    rq_activate_all_grippers(False)
    # end: URCap Program Node
    $ 4 "MoveJ"
    $ 5 "Waypoint_2" "breakAfter"
    movej(get_inverse_kin(Waypoint_2_p, qnear=Waypoint_2_q), a=1.3962634015954636, v=1.0471975511965976)
    $ 6 "Wait sensor=LO"
    while (get_standard_digital_in(0) == True):
      sync()
    end
    $ 7 "Pallet_1"
    def Pallet_1_trans(pose):
    return p[pose[0], pose[1], pose[2], 0, 0, 0]
  end
  def Pallet_1_rot(pose):
  return p[0, 0, 0, pose[3], pose[4], pose[5]]
  end
  def Pallet_1_compute_pallet_waypoint(T_base_feature_taught, T_feature_referencePoint_taught, T_referencePoint_approach_taught, T_base_feature, T_base_referencePoint):
  local trans_referencePoint_approach_in_feature_taught = pose_sub(Pallet_1_trans(pose_trans(T_feature_referencePoint_taught, T_referencePoint_approach_taught)), Pallet_1_trans(T_feature_referencePoint_taught))
  local rot_referencePoint_approach_in_feature_taught = pose_trans(Pallet_1_rot(T_feature_referencePoint_taught), pose_trans(Pallet_1_rot(T_referencePoint_approach_taught), pose_inv(Pallet_1_rot(T_feature_referencePoint_taught))))
  T_feature_referencePoint = pose_trans(pose_inv(T_base_feature), T_base_referencePoint)
  rot_referencePoint_approach = pose_trans(pose_inv(Pallet_1_rot(T_feature_referencePoint)), pose_trans(rot_referencePoint_approach_in_feature_taught, Pallet_1_rot(T_feature_referencePoint)))
  T_feature_approach = pose_trans(trans_referencePoint_approach_in_feature_taught, pose_trans(T_feature_referencePoint, rot_referencePoint_approach))
  T_base_approach = pose_trans(T_base_feature, T_feature_approach)
  return T_base_approach
  end
  Pallet_1_tct = 1
  if (Pallet_1_cnt_1 > 1 or Pallet_1_cnt_1 < 1):
    Pallet_1_cnt_1 = 1
  end
  $ 8 "Patterns" "noBreak"
  $ 9 "Irreg_Pattern_1" "noBreak"
  $ 11 "Layers" "noBreak"
  if (Pallet_1_cnt_1 < 2):
    Pallet_1_lno = 1
    Pallet_1_lct = Pallet_1_cnt_1
    global Item_1=pose_trans(p[0.0,0.0,0.0,0.0,0.0,0.0], pose_trans(p[-.000000000000, -.000000000000, -.000000000000, .000000000000, .000000000000, .000000000000], p[-.338171139538, -.420737183303, .092764235338, .009876315371, -3.096236515232, .249936558774]))
    if ((Pallet_1_lct - 1) == 0):
      referencePoint = Item_1
      Waypoint_6_q = [0.5956683158844361, -0.6755548280618635, 0.603014294320757, -1.6180516682204722, -1.4727962652724997, -0.9768632094038221]
    end
    direction = p[0,0,1,0,0,0]
    referencePoint = pose_add (referencePoint,p[0.0*direction[0],0.0*direction[1],0.0*direction[2],0,0,0])
  end
  Waypoint_6_p = Pallet_1_compute_pallet_waypoint(p[0.0,0.0,0.0,0.0,0.0,0.0], pose_trans(pose_inv(p[0.0,0.0,0.0,0.0,0.0,0.0]), p[-0.35656855679907695,-0.4237765193480358,0.0916497228884191,0.14229659831444877,-3.021243201222635,0.176167743332585]), p[-0.050081541706238464,-0.002934815571442262,-0.05522053959512324,0.06280827340026365,0.001341962689266323,0.110632066395465], p[0.0,0.0,0.0,0.0,0.0,0.0], referencePoint)
  Waypoint_6_p = pose_trans(p[-0.35656855679907695,-0.4237765193480358,0.0916497228884191,0.14229659831444882,-3.021243201222637,0.17616774333258506], pose_trans(pose_inv(referencePoint), Waypoint_6_p))
  Waypoint_7_p = Pallet_1_compute_pallet_waypoint(p[0.0,0.0,0.0,0.0,0.0,0.0], pose_trans(pose_inv(p[0.0,0.0,0.0,0.0,0.0,0.0]), p[-0.35656855679907695,-0.4237765193480358,0.0916497228884191,0.14229659831444877,-3.021243201222635,0.176167743332585]), p[-0.0972432192339368,0.006486004980699234,-0.006903856687141913,-0.09058990540327166,-0.07880304154291709,0.12847659139677955], p[0.0,0.0,0.0,0.0,0.0,0.0], referencePoint)
  Waypoint_7_p = pose_trans(p[-0.35656855679907695,-0.4237765193480358,0.0916497228884191,0.14229659831444882,-3.021243201222637,0.17616774333258506], pose_trans(pose_inv(referencePoint), Waypoint_7_p))
  Waypoint_6_p = Pallet_1_compute_pallet_waypoint(p[0.0,0.0,0.0,0.0,0.0,0.0], pose_trans(pose_inv(p[0.0,0.0,0.0,0.0,0.0,0.0]), p[-0.35656855679907695,-0.4237765193480358,0.0916497228884191,0.14229659831444877,-3.021243201222635,0.176167743332585]), p[-0.050081541706238464,-0.002934815571442262,-0.05522053959512324,0.06280827340026365,0.001341962689266323,0.110632066395465], p[0.0,0.0,0.0,0.0,0.0,0.0], referencePoint)
  Waypoint_6_p = pose_trans(p[-0.35656855679907695,-0.4237765193480358,0.0916497228884191,0.14229659831444882,-3.021243201222637,0.17616774333258506], pose_trans(pose_inv(referencePoint), Waypoint_6_p))
  $ 12 "At Each Item" "noBreak"
  $ 13 "Generated Movements" "noBreak"
  $ 14 "MoveJ" "noBreak"
  $ 15 "Waypoint_6" "noBreak"
  movej(get_inverse_kin(pose_trans(referencePoint, pose_trans(p[-.400294158776, .393560298227, .001491262390, -.142296598314, 3.021243201223, -.176167743333], Waypoint_6_p)), qnear=Waypoint_6_q), a=1.3962634015954636, v=1.0471975511965976)
  $ 16 "MoveL" "noBreak"
  $ 17 "Waypoint_7" "noBreak"
  movel(pose_trans(referencePoint, pose_trans(p[-.400294158776, .393560298227, .001491262390, -.142296598314, 3.021243201223, -.176167743333], Waypoint_7_p)), a=1.2, v=0.25)
  $ 18 "Set Payload: Payload" "noBreak"
  set_target_payload(0.450000, [0.000000, 0.000000, 0.000000], [0.000407, 0.000407, 0.000407, 0.000000, 0.000000, 0.000000])
  $ 19 "Tool action" "noBreak"
  # begin: URCap Program Node
  #   Source: Robotiq_Grippers, 2.4.0.45103, Robotiq Inc.
  #   Type: Gripper
  $ 20 "Gripper Close (3)" "noBreak"
  if not(gripper_connected[2]):
    popup("Gripper 3 must be connected to run this program.", "No connection", False, True, True)
  end
  if not(rq_is_gripper_activated("3")):
    popup("Gripper 3 is not activated. Go to Installation tab > Gripper to activate it and run the program again.", "Not activated", False, True, True)
  end
  rq_set_pos_spd_for(255, 255, 13, "3")
  rq_wait_pos_spe_for_request(255, 255, 13, "3")
  rq_go_to("3")
  rq_wait("3")
  # end: URCap Program Node
  $ 21 "MoveL" "noBreak"
  $ 22 "Waypoint_6" "noBreak"
  movel(pose_trans(referencePoint, pose_trans(p[-.400294158776, .393560298227, .001491262390, -.142296598314, 3.021243201223, -.176167743333], Waypoint_6_p)), a=1.2, v=0.25)
  Pallet_1_sep = False
  if (Pallet_1_cnt_1 >= 1):
    Pallet_1_cnt_1 = 1
  else:
    Pallet_1_cnt_1 = Pallet_1_cnt_1 + 1
  end
  $ 23 "Pallet_2"
  def Pallet_2_trans(pose):
  return p[pose[0], pose[1], pose[2], 0, 0, 0]
  end
  def Pallet_2_rot(pose):
  return p[0, 0, 0, pose[3], pose[4], pose[5]]
  end
  def Pallet_2_compute_pallet_waypoint(T_base_feature_taught, T_feature_referencePoint_taught, T_referencePoint_approach_taught, T_base_feature, T_base_referencePoint):
  local trans_referencePoint_approach_in_feature_taught = pose_sub(Pallet_2_trans(pose_trans(T_feature_referencePoint_taught, T_referencePoint_approach_taught)), Pallet_2_trans(T_feature_referencePoint_taught))
  local rot_referencePoint_approach_in_feature_taught = pose_trans(Pallet_2_rot(T_feature_referencePoint_taught), pose_trans(Pallet_2_rot(T_referencePoint_approach_taught), pose_inv(Pallet_2_rot(T_feature_referencePoint_taught))))
  T_feature_referencePoint = pose_trans(pose_inv(T_base_feature), T_base_referencePoint)
  rot_referencePoint_approach = pose_trans(pose_inv(Pallet_2_rot(T_feature_referencePoint)), pose_trans(rot_referencePoint_approach_in_feature_taught, Pallet_2_rot(T_feature_referencePoint)))
  T_feature_approach = pose_trans(trans_referencePoint_approach_in_feature_taught, pose_trans(T_feature_referencePoint, rot_referencePoint_approach))
  T_base_approach = pose_trans(T_base_feature, T_feature_approach)
  return T_base_approach
  end
  Pallet_2_tct = 1
  if (Pallet_2_cnt_1 > 1 or Pallet_2_cnt_1 < 1):
    Pallet_2_cnt_1 = 1
  end
  $ 24 "Patterns" "noBreak"
  $ 25 "Irreg_Pattern_2" "noBreak"
  $ 27 "Layers" "noBreak"
  if (Pallet_2_cnt_1 < 2):
    Pallet_2_lno = 1
    Pallet_2_lct = Pallet_2_cnt_1
    global Item_2=pose_trans(p[0.0,0.0,0.0,0.0,0.0,0.0], pose_trans(p[-.000000000000, -.000000000000, -.000000000000, .000000000000, .000000000000, .000000000000], p[-.463665534965, -.106220808801, .035787281560, 2.122926777319, 2.233821671100, -.100576269136]))
    if ((Pallet_2_lct - 1) == 0):
      referencePoin_1 = Item_2
      Waypoint_5_q = [-0.10132915178099822, -0.8465228837704926, 1.1239708105507988, -1.842076917673376, -1.4983623663589887, -0.15588361421827113]
    end
    direction = p[0,0,1,0,0,0]
    referencePoin_1 = pose_add (referencePoin_1,p[0.0*direction[0],0.0*direction[1],0.0*direction[2],0,0,0])
  end
  Waypoint_5_p = Pallet_2_compute_pallet_waypoint(p[0.0,0.0,0.0,0.0,0.0,0.0], pose_trans(pose_inv(p[0.0,0.0,0.0,0.0,0.0,0.0]), p[-0.4636655349654482,-0.10622080880105224,0.035787281559670425,2.1229267773186806,2.233821671099525,-0.10057626913611485]), p[0.0025464538946822213,0.007379050264824327,-0.053400380694234195,-0.03847629676856576,-0.00190489899378521,-0.0019139929032188495], p[0.0,0.0,0.0,0.0,0.0,0.0], referencePoin_1)
  Waypoint_5_p = pose_trans(p[-0.4636655349654482,-0.10622080880105224,0.035787281559670425,2.122926777318679,2.233821671099524,-0.10057626913611215], pose_trans(pose_inv(referencePoin_1), Waypoint_5_p))
  ToolActionPoi_1_p = Pallet_2_compute_pallet_waypoint(p[0.0,0.0,0.0,0.0,0.0,0.0], pose_trans(pose_inv(p[0.0,0.0,0.0,0.0,0.0,0.0]), p[-0.4636655349654482,-0.10622080880105224,0.035787281559670425,2.1229267773186806,2.233821671099525,-0.10057626913611485]), p[0.0,5.551115123125783E-17,2.7755575615628914E-17,-2.567396382296971E-12,1.8025025916301725E-12,-1.5242017175308427E-12], p[0.0,0.0,0.0,0.0,0.0,0.0], referencePoin_1)
  ToolActionPoi_1_p = pose_trans(p[-0.4636655349654482,-0.10622080880105224,0.035787281559670425,2.122926777318679,2.233821671099524,-0.10057626913611215], pose_trans(pose_inv(referencePoin_1), ToolActionPoi_1_p))
  Waypoint_5_p = Pallet_2_compute_pallet_waypoint(p[0.0,0.0,0.0,0.0,0.0,0.0], pose_trans(pose_inv(p[0.0,0.0,0.0,0.0,0.0,0.0]), p[-0.4636655349654482,-0.10622080880105224,0.035787281559670425,2.1229267773186806,2.233821671099525,-0.10057626913611485]), p[0.0025464538946822213,0.007379050264824327,-0.053400380694234195,-0.03847629676856576,-0.00190489899378521,-0.0019139929032188495], p[0.0,0.0,0.0,0.0,0.0,0.0], referencePoin_1)
  Waypoint_5_p = pose_trans(p[-0.4636655349654482,-0.10622080880105224,0.035787281559670425,2.122926777318679,2.233821671099524,-0.10057626913611215], pose_trans(pose_inv(referencePoin_1), Waypoint_5_p))
  $ 28 "At Each Item" "noBreak"
  $ 29 "Generated Movements" "noBreak"
  $ 30 "MoveJ" "noBreak"
  $ 31 "Waypoint_5" "noBreak"
  movej(get_inverse_kin(pose_trans(referencePoin_1, pose_trans(p[.085151670364, .468686561658, .025128032432, -2.122926777319, -2.233821671100, .100576269136], Waypoint_5_p)), qnear=Waypoint_5_q), a=1.3962634015954636, v=1.0471975511965976)
  $ 32 "MoveL" "noBreak"
  $ 33 "ToolActionPoi_1" "noBreak"
  movel(pose_trans(referencePoin_1, pose_trans(p[.085151670364, .468686561658, .025128032432, -2.122926777319, -2.233821671100, .100576269136], ToolActionPoi_1_p)), a=1.2, v=0.25)
  $ 34 "Tool action" "noBreak"
  # begin: URCap Program Node
  #   Source: Robotiq_Grippers, 2.4.0.45103, Robotiq Inc.
  #   Type: Gripper
  $ 35 "Gripper Open (3)" "noBreak"
  if not(gripper_connected[2]):
    popup("Gripper 3 must be connected to run this program.", "No connection", False, True, True)
  end
  if not(rq_is_gripper_activated("3")):
    popup("Gripper 3 is not activated. Go to Installation tab > Gripper to activate it and run the program again.", "Not activated", False, True, True)
  end
  rq_set_pos_spd_for(0, 255, 255, "3")
  rq_wait_pos_spe_for_request(0, 255, 255, "3")
  rq_go_to("3")
  rq_wait("3")
  # end: URCap Program Node
  $ 36 "MoveL" "noBreak"
  $ 37 "Waypoint_5" "noBreak"
  movel(pose_trans(referencePoin_1, pose_trans(p[.085151670364, .468686561658, .025128032432, -2.122926777319, -2.233821671100, .100576269136], Waypoint_5_p)), a=1.2, v=0.25)
  Pallet_2_sep = False
  if (Pallet_2_cnt_1 >= 1):
    Pallet_2_cnt_1 = 1
  else:
    Pallet_2_cnt_1 = Pallet_2_cnt_1 + 1
  end
  $ 38 "MoveL"
  $ 39 "Waypoint_1" "breakAfter"
  movel(Waypoint_1_p, a=1.2, v=0.25)
  $ 40 "Wait: 3.0"
  sleep(3.0)
  $ 41 "Pallet_3"
  def Pallet_3_trans(pose):
  return p[pose[0], pose[1], pose[2], 0, 0, 0]
  end
  def Pallet_3_rot(pose):
  return p[0, 0, 0, pose[3], pose[4], pose[5]]
  end
  def Pallet_3_compute_pallet_waypoint(T_base_feature_taught, T_feature_referencePoint_taught, T_referencePoint_approach_taught, T_base_feature, T_base_referencePoint):
  local trans_referencePoint_approach_in_feature_taught = pose_sub(Pallet_3_trans(pose_trans(T_feature_referencePoint_taught, T_referencePoint_approach_taught)), Pallet_3_trans(T_feature_referencePoint_taught))
  local rot_referencePoint_approach_in_feature_taught = pose_trans(Pallet_3_rot(T_feature_referencePoint_taught), pose_trans(Pallet_3_rot(T_referencePoint_approach_taught), pose_inv(Pallet_3_rot(T_feature_referencePoint_taught))))
  T_feature_referencePoint = pose_trans(pose_inv(T_base_feature), T_base_referencePoint)
  rot_referencePoint_approach = pose_trans(pose_inv(Pallet_3_rot(T_feature_referencePoint)), pose_trans(rot_referencePoint_approach_in_feature_taught, Pallet_3_rot(T_feature_referencePoint)))
  T_feature_approach = pose_trans(trans_referencePoint_approach_in_feature_taught, pose_trans(T_feature_referencePoint, rot_referencePoint_approach))
  T_base_approach = pose_trans(T_base_feature, T_feature_approach)
  return T_base_approach
  end
  Pallet_2_tct_1 = 1
  if (Pallet_2_cnt_2 > 1 or Pallet_2_cnt_2 < 1):
    Pallet_2_cnt_2 = 1
  end
  $ 42 "Patterns" "noBreak"
  $ 43 "Irreg_Pattern_3" "noBreak"
  $ 45 "Layers" "noBreak"
  if (Pallet_2_cnt_2 < 2):
    Pallet_2_lno_1 = 1
    Pallet_2_lct_1 = Pallet_2_cnt_2
    global Item_3=pose_trans(p[0.0,0.0,0.0,0.0,0.0,0.0], pose_trans(p[-.000000000000, -.000000000000, -.000000000000, .000000000000, .000000000000, .000000000000], p[-.463665534965, -.106220808801, .035787281560, 2.122926777319, 2.233821671100, -.100576269136]))
    if ((Pallet_2_lct_1 - 1) == 0):
      referencePoin_2 = Item_3
      Waypoint_5_q = [-0.10132915178099822, -0.8465228837704926, 1.1239708105507988, -1.842076917673376, -1.4983623663589887, -0.15588361421827113]
    end
    direction = p[0,0,1,0,0,0]
    referencePoin_2 = pose_add (referencePoin_2,p[0.0*direction[0],0.0*direction[1],0.0*direction[2],0,0,0])
  end
  Waypoint_5_p = Pallet_3_compute_pallet_waypoint(p[0.0,0.0,0.0,0.0,0.0,0.0], pose_trans(pose_inv(p[0.0,0.0,0.0,0.0,0.0,0.0]), p[-0.4636655349654482,-0.10622080880105224,0.035787281559670425,2.1229267773186806,2.233821671099525,-0.10057626913611485]), p[0.0025464538946822213,0.007379050264824327,-0.053400380694234195,-0.03847629676856576,-0.00190489899378521,-0.0019139929032188495], p[0.0,0.0,0.0,0.0,0.0,0.0], referencePoin_2)
  Waypoint_5_p = pose_trans(p[-0.4636655349654482,-0.10622080880105224,0.035787281559670425,2.122926777318679,2.233821671099524,-0.10057626913611215], pose_trans(pose_inv(referencePoin_2), Waypoint_5_p))
  ToolActionPoi_1_p = Pallet_3_compute_pallet_waypoint(p[0.0,0.0,0.0,0.0,0.0,0.0], pose_trans(pose_inv(p[0.0,0.0,0.0,0.0,0.0,0.0]), p[-0.4636655349654482,-0.10622080880105224,0.035787281559670425,2.1229267773186806,2.233821671099525,-0.10057626913611485]), p[0.0,5.551115123125783E-17,2.7755575615628914E-17,-2.567396382296971E-12,1.8025025916301725E-12,-1.5242017175308427E-12], p[0.0,0.0,0.0,0.0,0.0,0.0], referencePoin_2)
  ToolActionPoi_1_p = pose_trans(p[-0.4636655349654482,-0.10622080880105224,0.035787281559670425,2.122926777318679,2.233821671099524,-0.10057626913611215], pose_trans(pose_inv(referencePoin_2), ToolActionPoi_1_p))
  Waypoint_5_p = Pallet_3_compute_pallet_waypoint(p[0.0,0.0,0.0,0.0,0.0,0.0], pose_trans(pose_inv(p[0.0,0.0,0.0,0.0,0.0,0.0]), p[-0.4636655349654482,-0.10622080880105224,0.035787281559670425,2.1229267773186806,2.233821671099525,-0.10057626913611485]), p[0.0025464538946822213,0.007379050264824327,-0.053400380694234195,-0.03847629676856576,-0.00190489899378521,-0.0019139929032188495], p[0.0,0.0,0.0,0.0,0.0,0.0], referencePoin_2)
  Waypoint_5_p = pose_trans(p[-0.4636655349654482,-0.10622080880105224,0.035787281559670425,2.122926777318679,2.233821671099524,-0.10057626913611215], pose_trans(pose_inv(referencePoin_2), Waypoint_5_p))
  $ 46 "At Each Item" "noBreak"
  $ 47 "Generated Movements" "noBreak"
  $ 48 "MoveJ" "noBreak"
  $ 49 "Waypoint_5" "noBreak"
  movej(get_inverse_kin(pose_trans(referencePoin_2, pose_trans(p[.085151670364, .468686561658, .025128032432, -2.122926777319, -2.233821671100, .100576269136], Waypoint_5_p)), qnear=Waypoint_5_q), a=1.3962634015954636, v=1.0471975511965976)
  $ 50 "MoveL" "noBreak"
  $ 51 "ToolActionPoi_1" "noBreak"
  movel(pose_trans(referencePoin_2, pose_trans(p[.085151670364, .468686561658, .025128032432, -2.122926777319, -2.233821671100, .100576269136], ToolActionPoi_1_p)), a=1.2, v=0.25)
  $ 52 "Tool action" "noBreak"
  # begin: URCap Program Node
  #   Source: Robotiq_Grippers, 2.4.0.45103, Robotiq Inc.
  #   Type: Gripper
  $ 53 "Gripper Close (3)" "noBreak"
  if not(gripper_connected[2]):
    popup("Gripper 3 must be connected to run this program.", "No connection", False, True, True)
  end
  if not(rq_is_gripper_activated("3")):
    popup("Gripper 3 is not activated. Go to Installation tab > Gripper to activate it and run the program again.", "Not activated", False, True, True)
  end
  rq_set_pos_spd_for(255, 255, 13, "3")
  rq_wait_pos_spe_for_request(255, 255, 13, "3")
  rq_go_to("3")
  rq_wait("3")
  # end: URCap Program Node
  $ 54 "MoveL" "noBreak"
  $ 55 "Waypoint_5" "noBreak"
  movel(pose_trans(referencePoin_2, pose_trans(p[.085151670364, .468686561658, .025128032432, -2.122926777319, -2.233821671100, .100576269136], Waypoint_5_p)), a=1.2, v=0.25)
  Pallet_2_sep_1 = False
  if (Pallet_2_cnt_2 >= 1):
    Pallet_2_cnt_2 = 1
  else:
    Pallet_2_cnt_2 = Pallet_2_cnt_2 + 1
  end
  $ 56 "MoveL"
  $ 57 "Waypoint_3" "breakAfter"
  movel(Waypoint_3_p, a=1.2, v=0.25)
  $ 58 "Pallet_4"
  def Pallet_4_trans(pose):
  return p[pose[0], pose[1], pose[2], 0, 0, 0]
  end
  def Pallet_4_rot(pose):
  return p[0, 0, 0, pose[3], pose[4], pose[5]]
  end
  def Pallet_4_compute_pallet_waypoint(T_base_feature_taught, T_feature_referencePoint_taught, T_referencePoint_approach_taught, T_base_feature, T_base_referencePoint):
  local trans_referencePoint_approach_in_feature_taught = pose_sub(Pallet_4_trans(pose_trans(T_feature_referencePoint_taught, T_referencePoint_approach_taught)), Pallet_4_trans(T_feature_referencePoint_taught))
  local rot_referencePoint_approach_in_feature_taught = pose_trans(Pallet_4_rot(T_feature_referencePoint_taught), pose_trans(Pallet_4_rot(T_referencePoint_approach_taught), pose_inv(Pallet_4_rot(T_feature_referencePoint_taught))))
  T_feature_referencePoint = pose_trans(pose_inv(T_base_feature), T_base_referencePoint)
  rot_referencePoint_approach = pose_trans(pose_inv(Pallet_4_rot(T_feature_referencePoint)), pose_trans(rot_referencePoint_approach_in_feature_taught, Pallet_4_rot(T_feature_referencePoint)))
  T_feature_approach = pose_trans(trans_referencePoint_approach_in_feature_taught, pose_trans(T_feature_referencePoint, rot_referencePoint_approach))
  T_base_approach = pose_trans(T_base_feature, T_feature_approach)
  return T_base_approach
  end
  Pallet_4_tct = 6
  if (Pallet_4_cnt > 6 or Pallet_4_cnt < 1):
    Pallet_4_cnt = 1
  end
  $ 59 "Patterns" "noBreak"
  $ 60 "Grid_Pattern_1" "noBreak"
  $ 65 "Layers" "noBreak"
  if (Pallet_4_cnt < 7):
    Pallet_4_lno = 1
    Pallet_4_lct = Pallet_4_cnt
    global CornerItem_1=pose_trans(p[0.0,0.0,0.0,0.0,0.0,0.0], pose_trans(p[-.000000000000, -.000000000000, -.000000000000, .000000000000, .000000000000, .000000000000], p[.382936219048, -.260937906153, .035431334582, 3.123820532524, -.026843373394, .048126287698]))
    global CornerItem_2=pose_trans(p[0.0,0.0,0.0,0.0,0.0,0.0], pose_trans(p[-.000000000000, -.000000000000, -.000000000000, .000000000000, .000000000000, .000000000000], p[.381335191349, -.070417828845, .025325712282, -3.136237899403, .016530215479, .025476655283]))
    global CornerItem_3=pose_trans(p[0.0,0.0,0.0,0.0,0.0,0.0], pose_trans(p[-.000000000000, -.000000000000, -.000000000000, .000000000000, .000000000000, .000000000000], p[.492735594933, -.066091679299, .038035943765, 3.130149582825, -.084840850022, .029869593945]))
    global CornerItem_4=pose_trans(p[0.0,0.0,0.0,0.0,0.0,0.0], pose_trans(p[-.000000000000, -.000000000000, -.000000000000, .000000000000, .000000000000, .000000000000], p[.489230862545, -.252075252407, .033452933952, 3.079674293036, -.092801800985, .121199248000]))
    Pallet_4_cnt_x = (Pallet_4_lct - 1) % 2
    Pallet_4_cnt_y = floor((Pallet_4_lct - 1) / 2)
    referencePoin_3 = interpolate_pose(interpolate_pose(CornerItem_1, CornerItem_2, Pallet_4_cnt_x/1), interpolate_pose(CornerItem_4, CornerItem_3,Pallet_4_cnt_x/1), Pallet_4_cnt_y/2)
    direction = p[0,0,1,0,0,0]
    referencePoin_3 = pose_add (referencePoin_3,p[0.0*direction[0],0.0*direction[1],0.0*direction[2],0,0,0])
  end
  Approach_p = Pallet_4_compute_pallet_waypoint(p[0.0,0.0,0.0,0.0,0.0,0.0], pose_trans(pose_inv(p[0.0,0.0,0.0,0.0,0.0,0.0]), p[0.3689028710500054,-0.26596999301146235,0.036510209070372474,2.247353225191139,-2.156110811738366,-0.08527453507689232]), p[3.109304192189244E-4,0.0010672621443662544,-0.050637090985571745,0.03819688771906698,0.003411051993378327,0.044217408223267224], p[0.0,0.0,0.0,0.0,0.0,0.0], referencePoin_3)
  Approach_p = pose_trans(p[0.3689028710500054,-0.26596999301146235,0.036510209070372474,2.247353225191155,-2.156110811738381,-0.08527453507689652], pose_trans(pose_inv(referencePoin_3), Approach_p))
  Waypoint_4_p = Pallet_4_compute_pallet_waypoint(p[0.0,0.0,0.0,0.0,0.0,0.0], pose_trans(pose_inv(p[0.0,0.0,0.0,0.0,0.0,0.0]), p[0.3689028710500054,-0.26596999301146235,0.036510209070372474,2.247353225191139,-2.156110811738366,-0.08527453507689232]), p[0.003355513889856776,-0.010272763439174437,-0.011089809300880257,-0.03801218845341532,3.750061712264378E-4,0.004784064980047905], p[0.0,0.0,0.0,0.0,0.0,0.0], referencePoin_3)
  Waypoint_4_p = pose_trans(p[0.3689028710500054,-0.26596999301146235,0.036510209070372474,2.247353225191155,-2.156110811738381,-0.08527453507689652], pose_trans(pose_inv(referencePoin_3), Waypoint_4_p))
  Approach_p = Pallet_4_compute_pallet_waypoint(p[0.0,0.0,0.0,0.0,0.0,0.0], pose_trans(pose_inv(p[0.0,0.0,0.0,0.0,0.0,0.0]), p[0.3689028710500054,-0.26596999301146235,0.036510209070372474,2.247353225191139,-2.156110811738366,-0.08527453507689232]), p[3.109304192189244E-4,0.0010672621443662544,-0.050637090985571745,0.03819688771906698,0.003411051993378327,0.044217408223267224], p[0.0,0.0,0.0,0.0,0.0,0.0], referencePoin_3)
  Approach_p = pose_trans(p[0.3689028710500054,-0.26596999301146235,0.036510209070372474,2.247353225191155,-2.156110811738381,-0.08527453507689652], pose_trans(pose_inv(referencePoin_3), Approach_p))
  $ 66 "At Each Item" "noBreak"
  $ 67 "Generated Movements" "noBreak"
  $ 68 "MoveJ" "noBreak"
  $ 69 "Approach" "noBreak"
  movej(get_inverse_kin(pose_trans(referencePoin_3, pose_trans(p[-.279956932091, .354754852525, .062733337246, -2.247353225191, 2.156110811738, .085274535077], Approach_p)), qnear=Approach_q), a=1.3962634015954636, v=1.0471975511965976)
  $ 70 "MoveL" "noBreak"
  $ 71 "Waypoint_4" "noBreak"
  movel(pose_trans(referencePoin_3, pose_trans(p[-.279956932091, .354754852525, .062733337246, -2.247353225191, 2.156110811738, .085274535077], Waypoint_4_p)), a=1.2, v=0.25)
  $ 72 "Tool action" "noBreak"
  # begin: URCap Program Node
  #   Source: Robotiq_Grippers, 2.4.0.45103, Robotiq Inc.
  #   Type: Gripper
  $ 73 "Gripper Open (3)" "noBreak"
  if not(gripper_connected[2]):
    popup("Gripper 3 must be connected to run this program.", "No connection", False, True, True)
  end
  if not(rq_is_gripper_activated("3")):
    popup("Gripper 3 is not activated. Go to Installation tab > Gripper to activate it and run the program again.", "Not activated", False, True, True)
  end
  rq_set_pos_spd_for(0, 255, 255, "3")
  rq_wait_pos_spe_for_request(0, 255, 255, "3")
  rq_go_to("3")
  rq_wait("3")
  # end: URCap Program Node
  $ 74 "MoveL" "noBreak"
  $ 75 "Approach" "noBreak"
  movel(pose_trans(referencePoin_3, pose_trans(p[-.279956932091, .354754852525, .062733337246, -2.247353225191, 2.156110811738, .085274535077], Approach_p)), a=1.2, v=0.25)
  Pallet_4_sep = False
  if (Pallet_4_cnt >= 6):
    Pallet_4_cnt = 1
  else:
    Pallet_4_cnt = Pallet_4_cnt + 1
  end
  end
end
